PROGRAM FertilizerProcess
VAR

(***********************************************Napedy w procesie produkcji nawozu z pofermentu i osadu****************************************************************************************)
	//Napedy U11 pompy SP02	
	fbDrvInv_SP02 		: FB_DriveInv(1, E_InvType.Schneider);
	fbDrvContrInv_SP02  : FB_DriveControl(fbDrvInv_SP02);

	//Napedy M01 M02 VR01 - schemat U71, U81	
	fbDrvInv_M01 		: FB_DriveInv(7, E_InvType.Schneider);
	fbDrvContrInv_M01   : FB_DriveControl(fbDrvInv_M01);
	
	fbDrvInv_M02 		: FB_DriveInv(8, E_InvType.Schneider);
	fbDrvContrInv_M02   : FB_DriveControl(fbDrvInv_M02);
	
	//Naped klapy M03 VR01 - schemat U91 
	fbDrvInv_M03 		: FB_DriveInv(9, E_InvType.Schneider);
	fbDrvContrInv_M03   : FB_DriveControl(fbDrvInv_M03);
	
	//Naped wentylator BL01
	fbDrv_BL01			: FB_Drive_1C();
	fbDrvContr_BL01		: FB_DriveControl(fbDrv_BL01);

	//Napedy podajnik SC-01 i SC02
	fbDrv_SC01			: FB_Drive_1C();
	fbDrvContr_SC01	    : FB_DriveControl(fbDrv_SC01);
	
	fbDrv_SC02			: FB_Drive_1C();
	fbDrvContr_SC02		: FB_DriveControl(fbDrv_SC02);
		
	//Napedy S01_E01 i S02_E02
	fbDrv_E01			: FB_Drive_1C();
	fbDrvContr_E01	    : FB_DriveControl(fbDrv_E01);
	
	fbDrv_E02			: FB_Drive_1C();
	fbDrvContr_E02		: FB_DriveControl(fbDrv_E02);
	


(***********************************************Czujniki w procesie produkcji nawozu z pofermentu i osadu****************************************************************************************)
	//Temp Sensor
	fbTempSens_H01	 	: FB_Scaling; //Czujnik temperatury w hali H01
	
	//Rotary Sensor
	fbRotarySens_S01	 : FB_DigitalSensNC; //Czujnik poziomu w silosien S01 typu NC
	fbRotarySens_S02	 : FB_DigitalSensNC; //Czujnik poziomu w silosien S02 typu NC



(*********************************************** Bloki Process Controlller****************************************************************************************)

	(************** Granulation controller **************************************************)
	fbGranulationProcess : FB_GranulationProcess;
	
	(************** Flap controller **************************************************)
	fbFlapControl		: FB_FlapCtrl; //controller bloku sterowania klapa
	
	(************* Sludge dosing Controller ******************************************)
	fbSludgeDosing		: FB_SludgeDosing;
	
	(************ Manual Valve Position **********************************************)
	fbValvePosition_ZR01 : FB_DigitalSensNO;
	fbValvePosition_ZR02 : FB_DigitalSensNO;


	(****************** ZW02 - Przekaźnik K301 ******************************************************)
	fbContactor_ZW02	:	FB_Contactor(en:=GVL_Fertilizer.stContactor_ZW02.bCmd);
	
	(****************** H01 - Przekaźnik K303 ******************************************************)
	fbContactor_H01	:	FB_Contactor(en:=GVL_Cogeneration.stMixit_H01.Out); //uruchom wentylator gdy dziala mixit

	
	(****Filtr medianowy zakłoceń sygnałów analogowych**)
	fbMedian5_TempSens: FB_Median5;
	
	(*Detektor suchobiegu*)
	fbPumpDryRunDetector	: FB_PumpDryRunDetector;
END_VAR
VAR // added by the converter: edge detectors and wires of the graphical bodies
    _w1, _w2 : ANY;
END_VAR

//Action
//Czujniki
ACT_WeightSensor(); //Sensor wagowy
ACT_TempSens();		//Sensor temperatury
ACT_DigitalSens();  //Sensory poziomu

//Automat dozowania granulowania  i dozowania fermentacji
ACT_Control(); //Sterowanie procesem granulacji
ACT_SludgeDosing(); //sterowanie dozowaniem osadu do reaktora fermentacji R01


//Wybór nastawy napedów Auto lub SCADA
ACT_Motor(); //nastawy z SCADA

//Wykrywanie suchobiegu SP02
ACT_DryPumpDetection();



//**********************************SP-02*********************************************
//SP02
fbDrvContrInv_SP02();
GVL_Fertilizer.stDriveStatus_SP02 := fbDrvContrInv_SP02.StatusStruct(); //zwróc strukturę

//mode SP02
// 0 - ręka
// 1 - fermentacja
// 2 - granulacja
// 3 - konflikt zaworów

IF GVL_Fertilizer.ValvePosition_ZR01.bValue AND NOT GVL_Fertilizer.ValvePosition_ZR02.bValue THEN
    GVL_Fertilizer.iSP02_Mode := 1;

ELSIF GVL_Fertilizer.ValvePosition_ZR02.bValue AND NOT GVL_Fertilizer.ValvePosition_ZR01.bValue THEN
    GVL_Fertilizer.iSP02_Mode := 2;

ELSIF NOT GVL_Fertilizer.ValvePosition_ZR01.bValue AND NOT GVL_Fertilizer.ValvePosition_ZR02.bValue THEN
    GVL_Fertilizer.iSP02_Mode := 0;

ELSE
    GVL_Fertilizer.iSP02_Mode := 3;
END_IF;



//**********************************VR01*****************************************************
//M01
fbDrvContrInv_M01();
GVL_Fertilizer.stDriveStatus_M01 := fbDrvContrInv_M01.StatusStruct(); //zwróc strukturę
//M02
fbDrvContrInv_M02();
GVL_Fertilizer.stDriveStatus_M02 := fbDrvContrInv_M02.StatusStruct(); //zwróc strukturę
//M03
fbDrvContrInv_M03();
GVL_Fertilizer.stDriveStatus_M03 := fbDrvContrInv_M03.StatusStruct();

//**********************************Silosy S01 i S02*****************************************************
//SC01
fbDrvContr_SC01();
GVL_Fertilizer.stDriveStatus_SC01 := fbDrvContr_SC01.StatusStruct(); //zwróc strukturę
//SC02
fbDrvContr_SC02();
GVL_Fertilizer.stDriveStatus_SC02 := fbDrvContr_SC02.StatusStruct(); //zwróc strukturę
//E01
fbDrvContr_E01();
GVL_Fertilizer.stDriveStatus_E01 := fbDrvContr_E01.StatusStruct(); //zwróc strukturę
//E02
fbDrvContr_E02();
GVL_Fertilizer.stDriveStatus_E02 := fbDrvContr_E02.StatusStruct(); //zwróc strukturę

//**********************************BL01*****************************************************
//BL01
fbDrvContr_BL01();
GVL_Fertilizer.stDriveStatus_BL01 := fbDrvContr_BL01.StatusStruct(); //zwróc strukturę


//ZW02
fbContactor_ZW02();
GVL_Fertilizer.stContactor_ZW02.bOut	:=	fbContactor_ZW02.State; //zwróc stan

//H01 nagrzewnica wentylat
fbContactor_H01();
GVL_Fertilizer.stContactor_H01.bOut	:=	fbContactor_H01.State; //zwróc stan

ACTION ACT_Control:
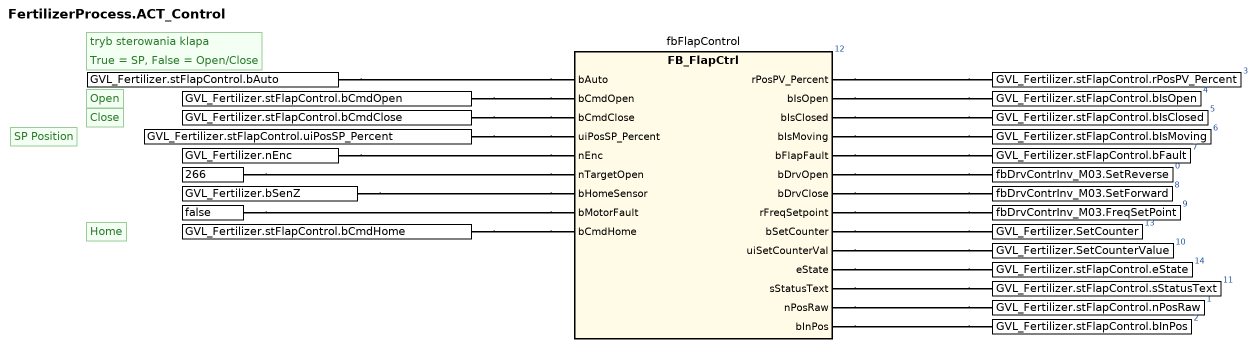
fbDrvContrInv_M03.SetReverse := fbFlapControl.bDrvOpen;
GVL_Fertilizer.stFlapControl.nPosRaw := fbFlapControl.nPosRaw;
GVL_Fertilizer.stFlapControl.bInPos := fbFlapControl.bInPos;
GVL_Fertilizer.stFlapControl.rPosPV_Percent := fbFlapControl.rPosPV_Percent;
GVL_Fertilizer.stFlapControl.bIsOpen := fbFlapControl.bIsOpen;
// Close
GVL_Fertilizer.stFlapControl.bIsClosed := fbFlapControl.bIsClosed;
// SP Position
GVL_Fertilizer.stFlapControl.bIsMoving := fbFlapControl.bIsMoving;
GVL_Fertilizer.stFlapControl.bFault := fbFlapControl.bFlapFault;
fbDrvContrInv_M03.SetForward := fbFlapControl.bDrvClose;
fbDrvContrInv_M03.FreqSetPoint := fbFlapControl.rFreqSetpoint;
GVL_Fertilizer.SetCounterValue := fbFlapControl.uiSetCounterVal;
GVL_Fertilizer.stFlapControl.sStatusText := fbFlapControl.sStatusText;
// tryb sterowania klapa
// True = SP, False = Open/Close
// Open
fbFlapControl(
    bAuto := GVL_Fertilizer.stFlapControl.bAuto,
    bCmdOpen := GVL_Fertilizer.stFlapControl.bCmdOpen,
    bCmdClose := GVL_Fertilizer.stFlapControl.bCmdClose,
    uiPosSP_Percent := GVL_Fertilizer.stFlapControl.uiPosSP_Percent,
    nEnc := GVL_Fertilizer.nEnc,
    nTargetOpen := 266,
    bHomeSensor := GVL_Fertilizer.bSenZ,
    bMotorFault := false,
    bCmdHome := GVL_Fertilizer.stFlapControl.bCmdHome); // FB_FlapCtrl
// Home
GVL_Fertilizer.SetCounter := fbFlapControl.bSetCounter;
GVL_Fertilizer.stFlapControl.eState := fbFlapControl.eState;
END_ACTION

ACTION ACT_DigitalSens:
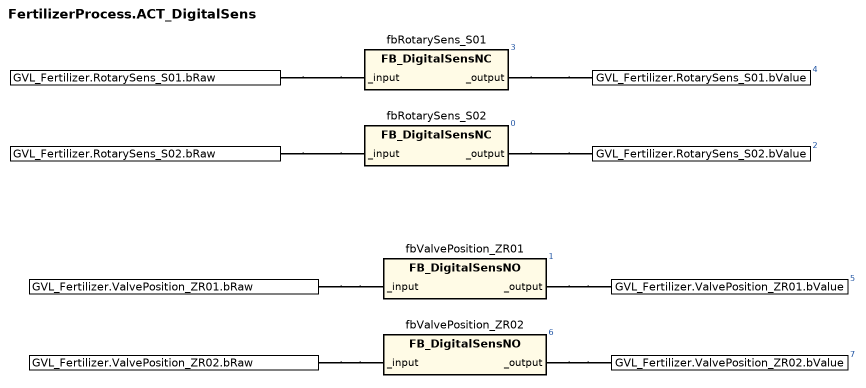
fbRotarySens_S02(_input := GVL_Fertilizer.RotarySens_S02.bRaw); // FB_DigitalSensNC
fbValvePosition_ZR01(_input := GVL_Fertilizer.ValvePosition_ZR01.bRaw); // FB_DigitalSensNO
GVL_Fertilizer.RotarySens_S02.bValue := fbRotarySens_S02._output;
fbRotarySens_S01(_input := GVL_Fertilizer.RotarySens_S01.bRaw); // FB_DigitalSensNC
GVL_Fertilizer.RotarySens_S01.bValue := fbRotarySens_S01._output;
GVL_Fertilizer.ValvePosition_ZR01.bValue := fbValvePosition_ZR01._output;
fbValvePosition_ZR02(_input := GVL_Fertilizer.ValvePosition_ZR02.bRaw); // FB_DigitalSensNO
GVL_Fertilizer.ValvePosition_ZR02.bValue := fbValvePosition_ZR02._output;
END_ACTION

ACTION ACT_DryPumpDetection:
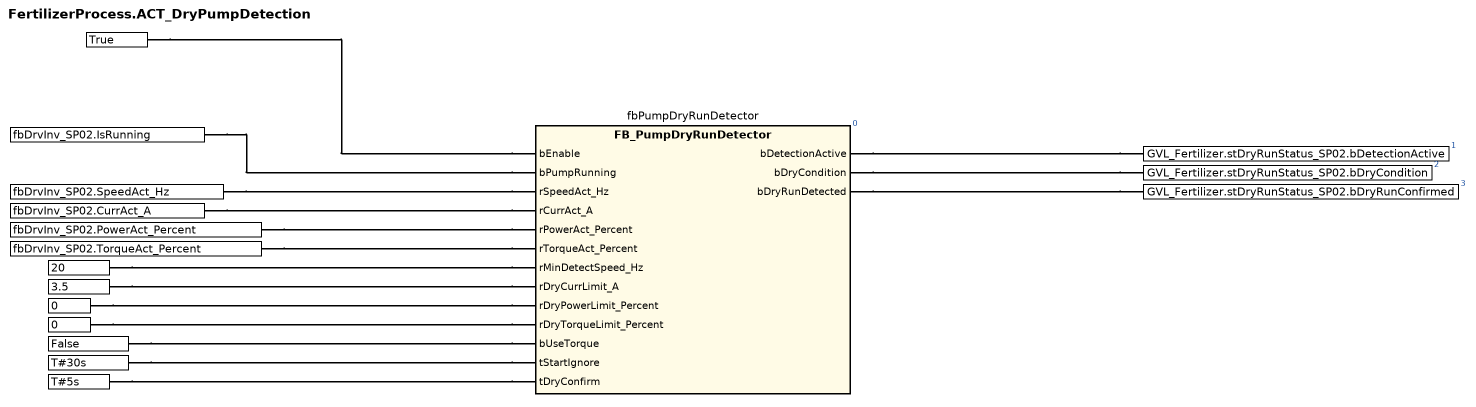
fbPumpDryRunDetector(
    bEnable := True,
    bPumpRunning := fbDrvInv_SP02.IsRunning,
    rSpeedAct_Hz := fbDrvInv_SP02.SpeedAct_Hz,
    rCurrAct_A := fbDrvInv_SP02.CurrAct_A,
    rPowerAct_Percent := fbDrvInv_SP02.PowerAct_Percent,
    rTorqueAct_Percent := fbDrvInv_SP02.TorqueAct_Percent,
    rMinDetectSpeed_Hz := 20,
    rDryCurrLimit_A := 3.5,
    rDryPowerLimit_Percent := 0,
    rDryTorqueLimit_Percent := 0,
    bUseTorque := False,
    tStartIgnore := T#30s,
    tDryConfirm := T#5s); // FB_PumpDryRunDetector
GVL_Fertilizer.stDryRunStatus_SP02.bDetectionActive := fbPumpDryRunDetector.bDetectionActive;
GVL_Fertilizer.stDryRunStatus_SP02.bDryCondition := fbPumpDryRunDetector.bDryCondition;
GVL_Fertilizer.stDryRunStatus_SP02.bDryRunConfirmed := fbPumpDryRunDetector.bDryRunDetected;
END_ACTION

ACTION ACT_Motor:

//************Naped ustawienia SP02**********************
//nastawy z SCADA lub z PLC blok nadrzędny wybór SELektorem
CASE GVL_Fertilizer.iSP02_Mode OF

    1: // FERMENTACJA
        fbDrvContrInv_SP02.SetForward   := fbSludgeDosing.bCmd_Pump;
        fbDrvContrInv_SP02.SetReverse   := FALSE;
        fbDrvContrInv_SP02.FreqSetPoint := fbSludgeDosing.rSpeedSet;

    2: // GRANULACJA
        fbDrvContrInv_SP02.SetForward   := fbGranulationProcess.bSP02_Fwd;
        fbDrvContrInv_SP02.SetReverse   := FALSE;
        fbDrvContrInv_SP02.FreqSetPoint := fbGranulationProcess.rSP02_Hz;

    0: // RĘKA
        fbDrvContrInv_SP02.SetForward   := GVL_Fertilizer.stDriveStatus_SP02.bForward;
        fbDrvContrInv_SP02.SetReverse   := GVL_Fertilizer.stDriveStatus_SP02.bReverse;
        fbDrvContrInv_SP02.FreqSetPoint := GVL_Fertilizer.stDriveStatus_SP02.FrequencySet;

    ELSE // KONFLIKT
        fbDrvContrInv_SP02.SetForward   := FALSE;
        fbDrvContrInv_SP02.SetReverse   := FALSE;
        fbDrvContrInv_SP02.FreqSetPoint := 0.0;
END_CASE;


//fbDrvContrInv_SP02.SetForward	:=SEL(fbGranulationProcess.bAutoTakeOver, GVL_Fertilizer.stDriveStatus_SP02.bForward, fbGranulationProcess.bSP02_Fwd);
//fbDrvContrInv_SP02.SetReverse	:=SEL(fbGranulationProcess.bAutoTakeOver, GVL_Fertilizer.stDriveStatus_SP02.bReverse, FALSE); // w automacie nie ma reverse
//fbDrvContrInv_SP02.FreqSetPoint	:=SEL(fbGranulationProcess.bAutoTakeOver, GVL_Fertilizer.stDriveStatus_SP02.FrequencySet, fbGranulationProcess.rSP02_Hz);

//***********Naped ustawienia VR01************************
//nastawy z SCADA M01 lub z PLC blok nadrzędny wybór SELektorem
fbDrvContrInv_M01.SetForward	:=SEL(fbGranulationProcess.bAutoTakeOver, GVL_Fertilizer.stDriveStatus_M01.bForward, fbGranulationProcess.bM01_Fwd);
fbDrvContrInv_M01.SetReverse	:=SEL(fbGranulationProcess.bAutoTakeOver, GVL_Fertilizer.stDriveStatus_M01.bReverse, FALSE);
fbDrvContrInv_M01.FreqSetPoint	:=SEL(fbGranulationProcess.bAutoTakeOver, GVL_Fertilizer.stDriveStatus_M01.FrequencySet, fbGranulationProcess.rMix_Hz);

//nastawy z SCADA M02 lub z PLC blok nadrzędny wybór SELektorem
fbDrvContrInv_M02.SetForward	:=SEL(fbGranulationProcess.bAutoTakeOver, GVL_Fertilizer.stDriveStatus_M02.bForward, fbGranulationProcess.bM02_Fwd);
fbDrvContrInv_M02.SetReverse	:=SEL(fbGranulationProcess.bAutoTakeOver, GVL_Fertilizer.stDriveStatus_M02.bReverse, FALSE);
fbDrvContrInv_M02.FreqSetPoint	:=SEL(fbGranulationProcess.bAutoTakeOver, GVL_Fertilizer.stDriveStatus_M02.FrequencySet, fbGranulationProcess.rMix_Hz);

//nastawy z SCADA M03
//fbDrvContrInv_M03.SetForward	:=GVL_Fertilizer.stDriveStatus_M03.bForward;
//fbDrvContrInv_M03.SetReverse	:=GVL_Fertilizer.stDriveStatus_M03.bReverse;
//fbDrvContrInv_M03.FreqSetPoint  :=GVL_Fertilizer.stDriveStatus_M03.FrequencySet;

//***********Naped ustawienia S01 i S02************************
//nastawy z SCADA SC01
fbDrvContr_SC01.SetForward	:=SEL(fbGranulationProcess.bAutoTakeOver, GVL_Fertilizer.stDriveStatus_SC01.bForward, fbGranulationProcess.bSC01_On);
//nastawy z SCADA SC02
fbDrvContr_SC02.SetForward	:=SEL(fbGranulationProcess.bAutoTakeOver, GVL_Fertilizer.stDriveStatus_SC02.bForward, fbGranulationProcess.bSC02_On);
//nastawy z SCADA E01
fbDrvContr_E01.SetForward	:=SEL(fbGranulationProcess.bAutoTakeOver, GVL_Fertilizer.stDriveStatus_E01.bForward, fbGranulationProcess.bE01_On);
//nastawy z SCADA E02
fbDrvContr_E02.SetForward	:=SEL(fbGranulationProcess.bAutoTakeOver, GVL_Fertilizer.stDriveStatus_E02.bForward, fbGranulationProcess.bE02_On);

////***********Naped ustawienia BL01 ************************
//nastawy z SCADA BL01
fbDrvContr_BL01.SetForward	:=SEL(fbGranulationProcess.bAutoTakeOver, GVL_Fertilizer.stDriveStatus_BL01.bForward, fbGranulationProcess.bBL01_On);
END_ACTION

ACTION ACT_SludgeDosing:
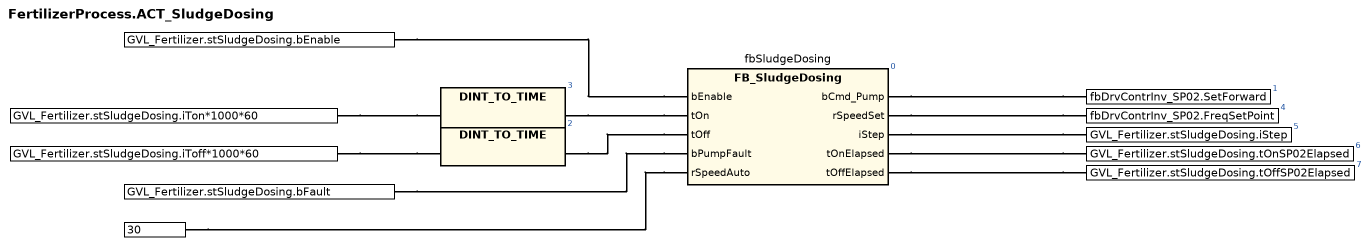
fbSludgeDosing(
    bEnable := GVL_Fertilizer.stSludgeDosing.bEnable,
    tOn := _w1,
    tOff := _w2,
    bPumpFault := GVL_Fertilizer.stSludgeDosing.bFault,
    rSpeedAuto := 30); // FB_SludgeDosing
fbDrvContrInv_SP02.SetForward := fbSludgeDosing.bCmd_Pump;
_w2 := DINT_TO_TIME(GVL_Fertilizer.stSludgeDosing.iToff*1000*60);
_w1 := DINT_TO_TIME(GVL_Fertilizer.stSludgeDosing.iTon*1000*60);
fbDrvContrInv_SP02.FreqSetPoint := fbSludgeDosing.rSpeedSet;
GVL_Fertilizer.stSludgeDosing.iStep := fbSludgeDosing.iStep;
GVL_Fertilizer.stSludgeDosing.tOnSP02Elapsed := fbSludgeDosing.tOnElapsed;
GVL_Fertilizer.stSludgeDosing.tOffSP02Elapsed := fbSludgeDosing.tOffElapsed;
END_ACTION

ACTION ACT_TempSens:
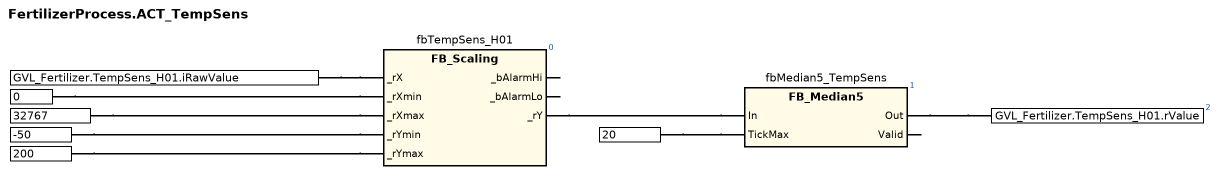
fbTempSens_H01(
    _rX := GVL_Fertilizer.TempSens_H01.iRawValue,
    _rXmin := 0,
    _rXmax := 32767,
    _rYmin := -50,
    _rYmax := 200); // FB_Scaling
fbMedian5_TempSens(In := fbTempSens_H01._rY, TickMax := 20); // FB_Median5
GVL_Fertilizer.TempSens_H01.rValue := fbMedian5_TempSens.Out;
END_ACTION

ACTION ACT_WeightSensor:
//******************************************** Weight 01 ****************************************************
// WORD jest ze znakiem więc najpierw konwertujemy na INt aby otrzymac znak a potem na REAL

GVL_Fertilizer.WeightSens_VR01.rWeightValue := TO_REAL(TO_INT(GVL_Fertilizer.WeightSens_VR01.rRawWeightValue));
END_ACTION

END_PROGRAM

(* stored: Version 1.1.0.1, ProductVersion 3.1.4024.16
   POU FertilizerProcess: Id {ae9cea5e-de76-4d67-bab9-1dcc1d16bc80}, SpecialFunc None
   Action ACT_Control: Id {c00a6ec6-8960-40d8-ac4d-33202791525f}
   Action ACT_DigitalSens: Id {90fd9b42-e3eb-4636-915c-8178b327b54f}
   Action ACT_DryPumpDetection: Id {0d630352-3f80-49b3-ae68-f847cc8845bd}
   Action ACT_Motor: Id {157fa111-0c10-4c74-bf66-984a77c8c761}
   Action ACT_SludgeDosing: Id {70e48efe-d9f6-4bfc-a5d3-1100a1c31cc2}
   Action ACT_TempSens: Id {e5be406b-b6a0-4f64-8c1c-50c0deca9433}
   Action ACT_WeightSensor: Id {c3ec4534-bc74-4a01-b06c-42e2c4179453} *)
